// Mitsubishi GX Works2 project: fbEx01   PLC: Q02/Q02H

PROGRAM MAIN
VAR
  자기_1 : 자기;
  자기_2 : 자기;
  자기_3 : 자기;
  인터록_1 : 인터록;
  인터록_2 : 인터록;
  카운터_1 : 업카운터;
  다운카운터_1 : 다운카운터;
  다운카운터_2 : 다운카운터;
  다운카운터_3 : 다운카운터;
END_VAR
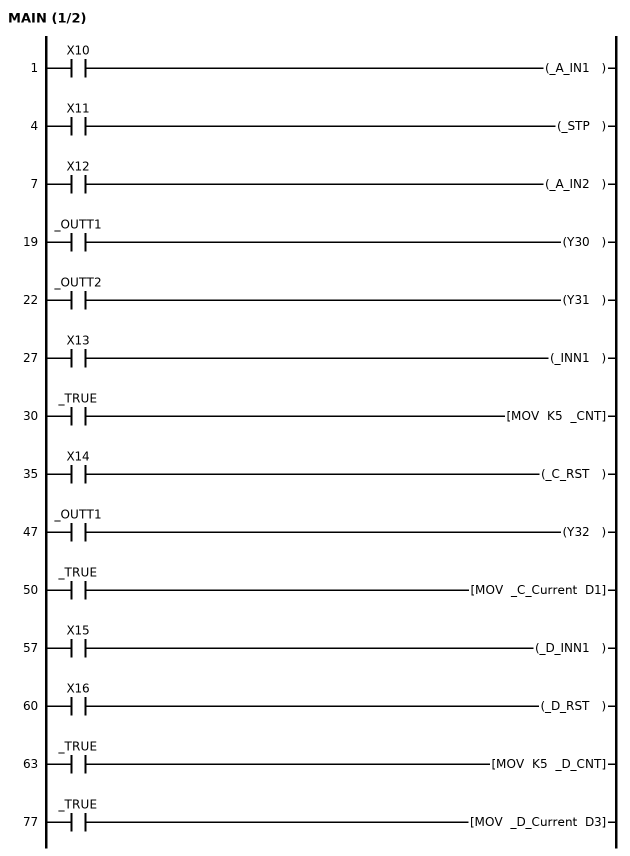
; FB BLK START 인터록(인터록_1)
1     LD      X10
      OUT     _A_IN1
4     LD      X11
      OUT     _STP
7     LD      X12
      OUT     _A_IN2
; FB START
; FB_NAME 인터록
; INSTANCE_NAME 인터록_1
; FB IN_B:A_IN1
; FB OUT_OUTT1:B
; FB IN_B:STP
; FB OUT_OUTT2:B
; FB IN_B:A_IN2
; FB END
19    LD      _OUTT1
      OUT     Y30
22    LD      _OUTT2
      OUT     Y31
; FB BLK END
; FB BLK START 업카운터(카운터_1)
27    LD      X13
      OUT     _INN1
30    LD      _TRUE
      MOV     K5 _CNT
35    LD      X14
      OUT     _C_RST
; FB START
; FB_NAME 업카운터
; INSTANCE_NAME 카운터_1
; FB IN_B:INN1
; FB OUT_OUTT1:B
; FB IN_W:CNT
; FB OUT_C_Current:W
; FB IN_B:C_RST
; FB END
47    LD      _OUTT1
      OUT     Y32
50    LD      _TRUE
      MOV     _C_Current D1
; FB BLK END
; FB BLK START 다운카운터(다운카운터_3)
57    LD      X15
      OUT     _D_INN1
60    LD      X16
      OUT     _D_RST
63    LD      _TRUE
      MOV     K5 _D_CNT
; FB START
; FB_NAME 다운카운터
; INSTANCE_NAME 다운카운터_3
; FB IN_B:D_INN1
; FB OUT_D_Current:W
; FB IN_B:D_RST
; FB OUT_D_OUTT1:B
; FB IN_W:D_CNT
; FB END
77    LD      _TRUE
      MOV     _D_Current D3
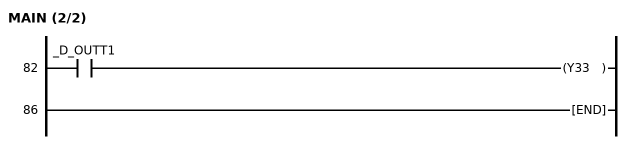
82    LD      _D_OUTT1
      OUT     Y33
; FB BLK END
86    END
END_PROGRAM

FUNCTION_BLOCK 자기
VAR_INPUT
  IN : BOOL;
END_VAR
VAR_OUTPUT
  OUTT : BOOL;
END_VAR
VAR_INPUT
  INN2 : BOOL;
END_VAR
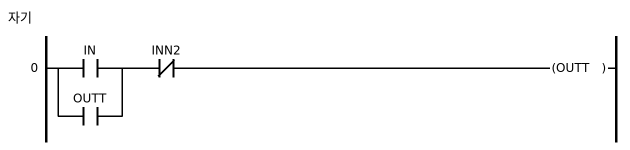
0     LD      IN
      OR      OUTT
      ANI     INN2
      OUT     OUTT
END_FUNCTION_BLOCK

FUNCTION_BLOCK 인터록
VAR_INPUT
  A_IN1 : BOOL;
  STP : BOOL;
END_VAR
VAR_OUTPUT
  OUTT1 : BOOL;
  OUTT2 : BOOL;
END_VAR
VAR_INPUT
  A_IN2 : BOOL;
END_VAR
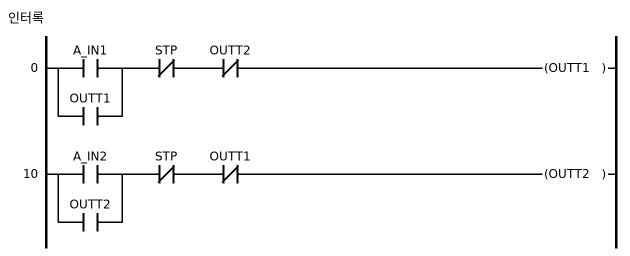
0     LD      A_IN1
      OR      OUTT1
      ANI     STP
      ANI     OUTT2
      OUT     OUTT1
10    LD      A_IN2
      OR      OUTT2
      ANI     STP
      ANI     OUTT1
      OUT     OUTT2
END_FUNCTION_BLOCK

FUNCTION_BLOCK 업카운터
VAR_INPUT
  INN1 : BOOL;
  CNT : INT;
  C_RST : BOOL;
END_VAR
VAR_OUTPUT
  OUTT1 : BOOL;
  C_Current : INT;
END_VAR
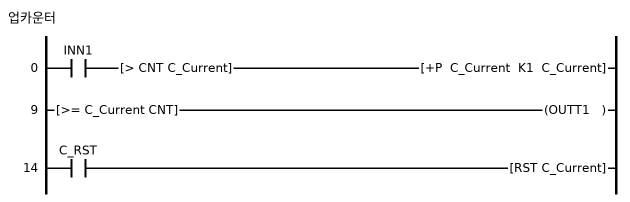
0     LD      INN1
      AND>    CNT C_Current
      +P      C_Current K1 C_Current
9     LD>=    C_Current CNT
      OUT     OUTT1
14    LD      C_RST
      RST     C_Current
END_FUNCTION_BLOCK

FUNCTION_BLOCK 다운카운터
VAR_OUTPUT
  D_Current : INT;
  D_OUTT1 : BOOL;
END_VAR
VAR_INPUT
  D_INN1 : BOOL;
  D_RST : BOOL;
  D_CNT : INT;
END_VAR
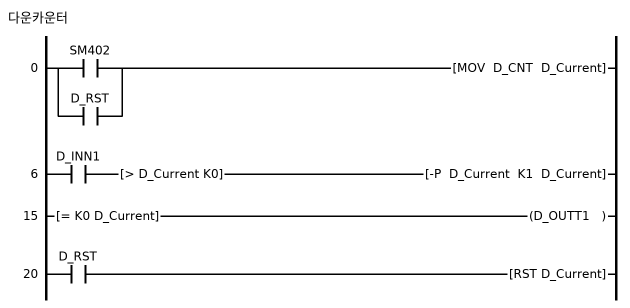
0     LD      SM402
      OR      D_RST
      MOV     D_CNT D_Current
6     LD      D_INN1
      AND>    D_Current K0
      -P      D_Current K1 D_Current
15    LD=     K0 D_Current
      OUT     D_OUTT1
20    LD      D_RST
      RST     D_Current
END_FUNCTION_BLOCK
